FUNCTION BOOLS_TO_BYTE
  (* Standard: 61499-1; Description: Copyright (c) 2024 HR Agrartechnik GmbH This program and the accompanying materials are made available under the terms of the Eclipse Public License 2.0 which is available at https://www.eclipse.org/legal/epl-2.0/ SPDX-License-Identifier: EPL-2.0 *)
  (* Version 1.0, 2024-02-22, franz *)
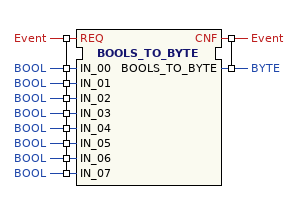
  EVENT_INPUT
    REQ WITH IN_00, IN_01, IN_02, IN_03, IN_04, IN_05, IN_06, IN_07;
  END_EVENT
  EVENT_OUTPUT
    CNF WITH BOOLS_TO_BYTE;
  END_EVENT
  VAR_INPUT
    IN_00 : BOOL; (* BIT 00 *)
    IN_01 : BOOL; (* BIT 01 *)
    IN_02 : BOOL; (* BIT 02 *)
    IN_03 : BOOL; (* BIT 03 *)
    IN_04 : BOOL; (* BIT 04 *)
    IN_05 : BOOL; (* BIT 05 *)
    IN_06 : BOOL; (* BIT 06 *)
    IN_07 : BOOL; (* BIT 07 *)
  END_VAR
  VAR_OUTPUT
    BOOLS_TO_BYTE : BYTE;
  END_VAR
  BODY IN ST:
FUNCTION BOOLS_TO_BYTE : BYTE

VAR_INPUT
	IN_00 : BOOL;    // BIT 00
	IN_01 : BOOL;    // BIT 01
	IN_02 : BOOL;    // BIT 02
	IN_03 : BOOL;    // BIT 03
	IN_04 : BOOL;    // BIT 04
	IN_05 : BOOL;    // BIT 05
	IN_06 : BOOL;    // BIT 06
	IN_07 : BOOL;    // BIT 07
END_VAR

(* this Function combines the 8 BOOLS to a byte *)
BOOLS_TO_BYTE.0 := IN_00;
BOOLS_TO_BYTE.1 := IN_01;
BOOLS_TO_BYTE.2 := IN_02;
BOOLS_TO_BYTE.3 := IN_03;
BOOLS_TO_BYTE.4 := IN_04;
BOOLS_TO_BYTE.5 := IN_05;
BOOLS_TO_BYTE.6 := IN_06;
BOOLS_TO_BYTE.7 := IN_07;

END_FUNCTION
  END_BODY
END_FUNCTION
